TYPE EtcSlaveBase_82538BE2 :
STRUCT
END_STRUCT
END_TYPE

(* stored: Version 1.2.0.0
   DUT EtcSlaveBase_82538BE2: Id {c17d8134-8acd-473b-88d8-c3039af4d15c} *)
